(* IEC 61131-3 sources: ATCMcontrol_Engineering/src/COM/softing/fc/CL/Libs/ATCM_IEC1131_3/table_34, 2 files *)

(* ---- rs.st ---- *)
(*[[
    UserURL= "ATCMFile:RS.htm"
]]*)
FUNCTION_BLOCK RS
VAR_INPUT
   S  : BOOL;
   R1 : BOOL;
END_VAR
VAR_OUTPUT
   Q1 : BOOL;
END_VAR

 Q1 := NOT R1 AND (S OR Q1);

END_FUNCTION_BLOCK

(* ---- sr.st ---- *)
(*[[
    UserURL= "ATCMFile:SR.htm"
]]*)
FUNCTION_BLOCK SR
VAR_INPUT
   S1 : BOOL;
   R  : BOOL;
END_VAR
VAR_OUTPUT
   Q1 : BOOL;
END_VAR

  Q1 := (NOT R AND Q1) OR S1;

END_FUNCTION_BLOCK
